% RSLogix 500 project project4.RSS, saved by version 8.30.00.16 %
PROJECT "UNTITLED"    % processor: Bul.1763 MicroLogix 1100 Series B %

PROGRAM FILES
  LAD 2 "MAIN"  4 rungs
  LAD 3 "DIGITAL IO"  7 rungs
  LAD 4 "CONTROLS"  13 rungs
  LAD 5 "MODES"  8 rungs

DATA FILES
  O0 OUTPUT  5 elements
  I1 INPUT  7 elements
  S2 STATUS  66 elements
  B3 BINARY  2 elements
  T4 TIMER  3 elements
  C5 COUNTER  1 elements
  R6 CONTROL  1 elements
  N7 INTEGER  2 elements
  F8 FLOAT  1 elements

LADDER 2 "MAIN"
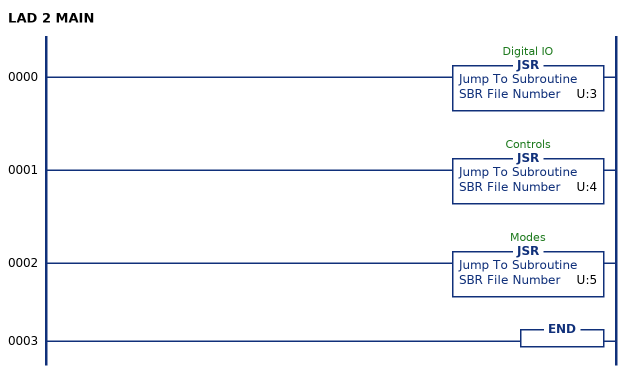
% Rung: 0 %
SOR JSR U:3 EOR
%   U:3  "Digital IO" %
% Rung: 1 %
SOR JSR U:4 EOR
%   U:4  "Controls" %
% Rung: 2 %
SOR JSR U:5 EOR
%   U:5  "Modes" %
% Rung: 3 %
SOR END EOR

LADDER 3 "DIGITAL IO"
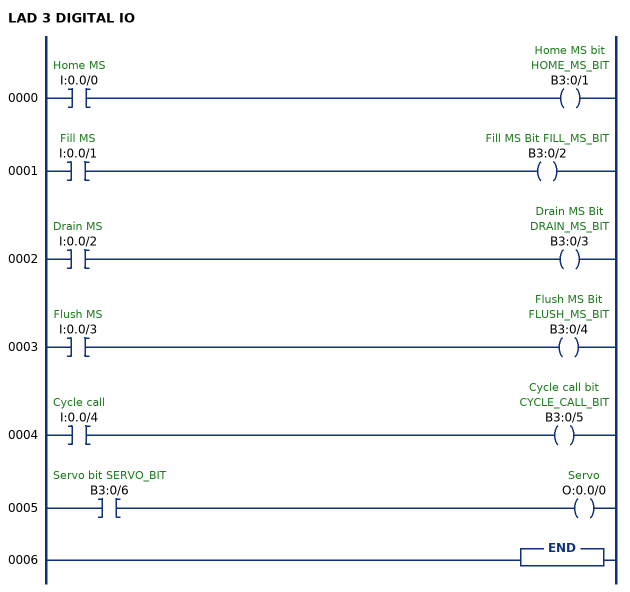
% Rung: 0 %
SOR XIC I:0.0/0 OTE B3:0/1 EOR
%   I:0.0/0  "Home MS" %
%   B3:0/1  HOME_MS_BIT  "Home MS bit" %
% Rung: 1 %
SOR XIC I:0.0/1 OTE B3:0/2 EOR
%   I:0.0/1  "Fill MS" %
%   B3:0/2  FILL_MS_BIT  "Fill MS Bit" %
% Rung: 2 %
SOR XIC I:0.0/2 OTE B3:0/3 EOR
%   I:0.0/2  "Drain MS" %
%   B3:0/3  DRAIN_MS_BIT  "Drain MS Bit" %
% Rung: 3 %
SOR XIC I:0.0/3 OTE B3:0/4 EOR
%   I:0.0/3  "Flush MS" %
%   B3:0/4  FLUSH_MS_BIT  "Flush MS Bit" %
% Rung: 4 %
SOR XIC I:0.0/4 OTE B3:0/5 EOR
%   I:0.0/4  "Cycle call" %
%   B3:0/5  CYCLE_CALL_BIT  "Cycle call bit" %
% Rung: 5 %
SOR XIC B3:0/6 OTE O:0.0/0 EOR
%   B3:0/6  SERVO_BIT  "Servo bit" %
%   O:0.0/0  "Servo" %
% Rung: 6 %
SOR END EOR

LADDER 4 "CONTROLS"
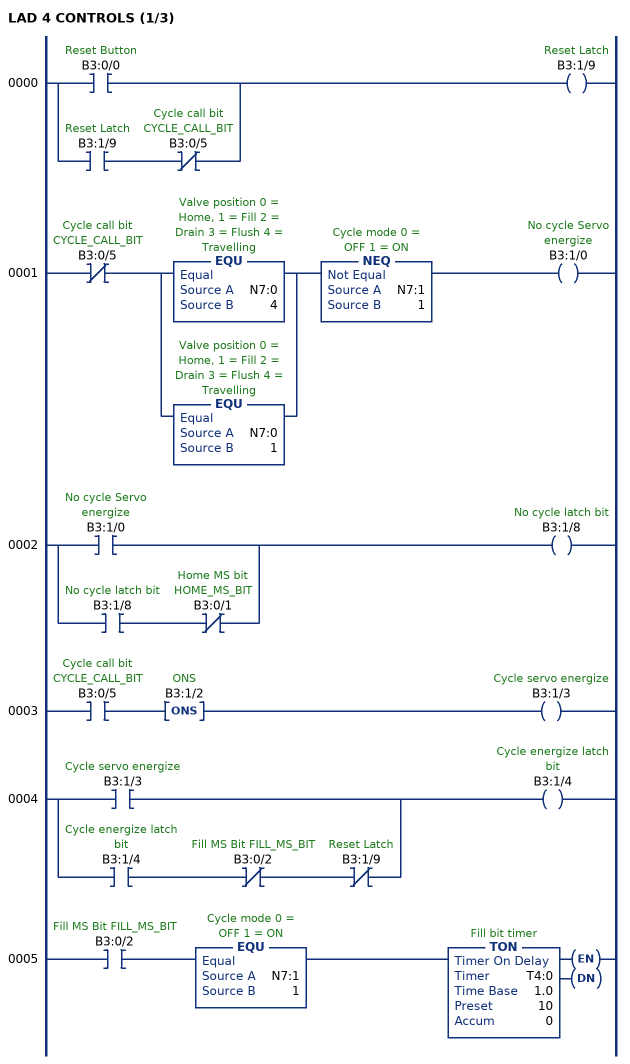
% Rung: 0 %
SOR BST XIC B3:0/0 NXB XIC B3:1/9 XIO B3:0/5 BND OTE B3:1/9 EOR
%   B3:0/0  "Reset Button" %
%   B3:1/9  "Reset Latch" %
%   B3:0/5  CYCLE_CALL_BIT  "Cycle call bit" %
% Rung: 1 %
SOR XIO B3:0/5 BST EQU N7:0 4 NXB EQU N7:0 1 BND NEQ N7:1 1 OTE B3:1/0 EOR
%   B3:0/5  CYCLE_CALL_BIT  "Cycle call bit" %
%   N7:0  "Valve position 0 = Home, 1 = Fill 2 = Drain 3 = Flush 4 = Travelling" %
%   N7:1  "Cycle mode 0 = OFF 1 = ON" %
%   B3:1/0  "No cycle Servo energize" %
% Rung: 2 %
SOR BST XIC B3:1/0 NXB XIC B3:1/8 XIO B3:0/1 BND OTE B3:1/8 EOR
%   B3:1/0  "No cycle Servo energize" %
%   B3:1/8  "No cycle latch bit" %
%   B3:0/1  HOME_MS_BIT  "Home MS bit" %
% Rung: 3 %
SOR XIC B3:0/5 ONS B3:1/2 OTE B3:1/3 EOR
%   B3:0/5  CYCLE_CALL_BIT  "Cycle call bit" %
%   B3:1/2  "ONS" %
%   B3:1/3  "Cycle servo energize" %
% Rung: 4 %
SOR BST XIC B3:1/3 NXB XIC B3:1/4 XIO B3:0/2 XIO B3:1/9 BND OTE B3:1/4 EOR
%   B3:1/3  "Cycle servo energize" %
%   B3:1/4  "Cycle energize latch bit" %
%   B3:0/2  FILL_MS_BIT  "Fill MS Bit" %
%   B3:1/9  "Reset Latch" %
% Rung: 5 %
SOR XIC B3:0/2 EQU N7:1 1 TON T4:0 1.0 10 0 EOR
%   B3:0/2  FILL_MS_BIT  "Fill MS Bit" %
%   N7:1  "Cycle mode 0 = OFF 1 = ON" %
%   T4:0  "Fill bit timer" %

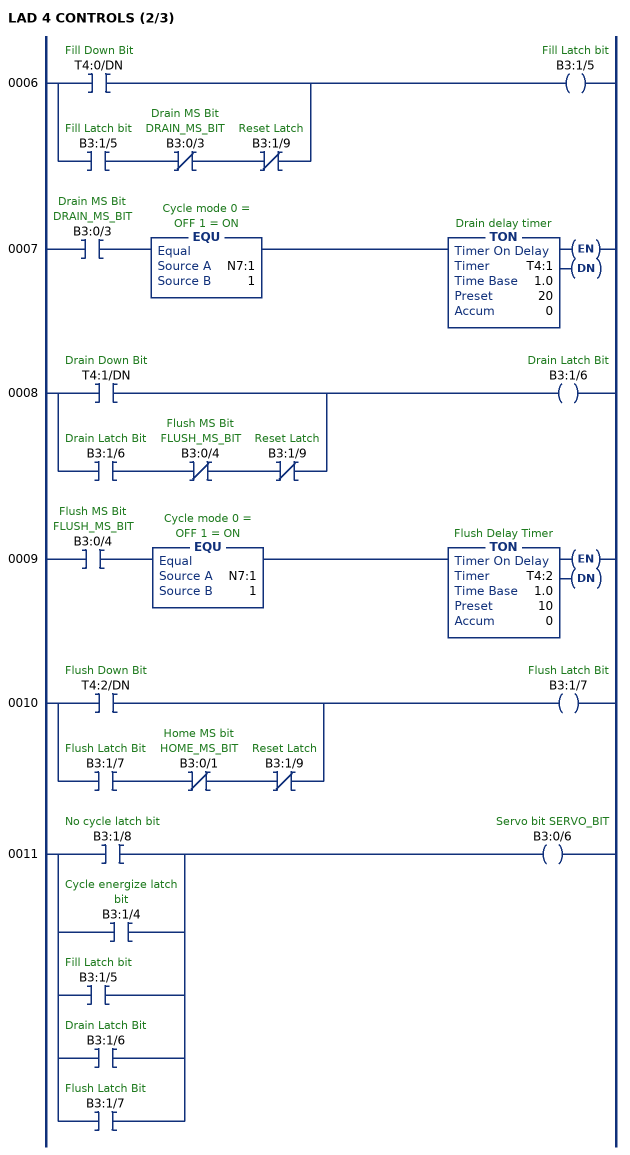
% Rung: 6 %
SOR BST XIC T4:0/DN NXB XIC B3:1/5 XIO B3:0/3 XIO B3:1/9 BND OTE B3:1/5 EOR
%   T4:0/DN  "Fill Down Bit" %
%   B3:1/5  "Fill Latch bit" %
%   B3:0/3  DRAIN_MS_BIT  "Drain MS Bit" %
%   B3:1/9  "Reset Latch" %
% Rung: 7 %
SOR XIC B3:0/3 EQU N7:1 1 TON T4:1 1.0 20 0 EOR
%   B3:0/3  DRAIN_MS_BIT  "Drain MS Bit" %
%   N7:1  "Cycle mode 0 = OFF 1 = ON" %
%   T4:1  "Drain delay timer" %
% Rung: 8 %
SOR BST XIC T4:1/DN NXB XIC B3:1/6 XIO B3:0/4 XIO B3:1/9 BND OTE B3:1/6 EOR
%   T4:1/DN  "Drain Down Bit" %
%   B3:1/6  "Drain Latch Bit" %
%   B3:0/4  FLUSH_MS_BIT  "Flush MS Bit" %
%   B3:1/9  "Reset Latch" %
% Rung: 9 %
SOR XIC B3:0/4 EQU N7:1 1 TON T4:2 1.0 10 0 EOR
%   B3:0/4  FLUSH_MS_BIT  "Flush MS Bit" %
%   N7:1  "Cycle mode 0 = OFF 1 = ON" %
%   T4:2  "Flush Delay Timer" %
% Rung: 10 %
SOR BST XIC T4:2/DN NXB XIC B3:1/7 XIO B3:0/1 XIO B3:1/9 BND OTE B3:1/7 EOR
%   T4:2/DN  "Flush Down Bit" %
%   B3:1/7  "Flush Latch Bit" %
%   B3:0/1  HOME_MS_BIT  "Home MS bit" %
%   B3:1/9  "Reset Latch" %
% Rung: 11 %
SOR BST XIC B3:1/8 NXB XIC B3:1/4 NXB XIC B3:1/5 NXB XIC B3:1/6 NXB XIC B3:1/7 BND OTE B3:0/6 EOR
%   B3:1/8  "No cycle latch bit" %
%   B3:1/4  "Cycle energize latch bit" %
%   B3:1/5  "Fill Latch bit" %
%   B3:1/6  "Drain Latch Bit" %
%   B3:1/7  "Flush Latch Bit" %
%   B3:0/6  SERVO_BIT  "Servo bit" %

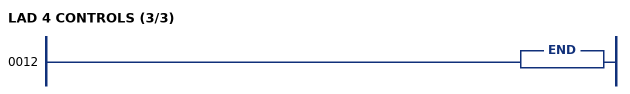
% Rung: 12 %
SOR END EOR

LADDER 5 "MODES"
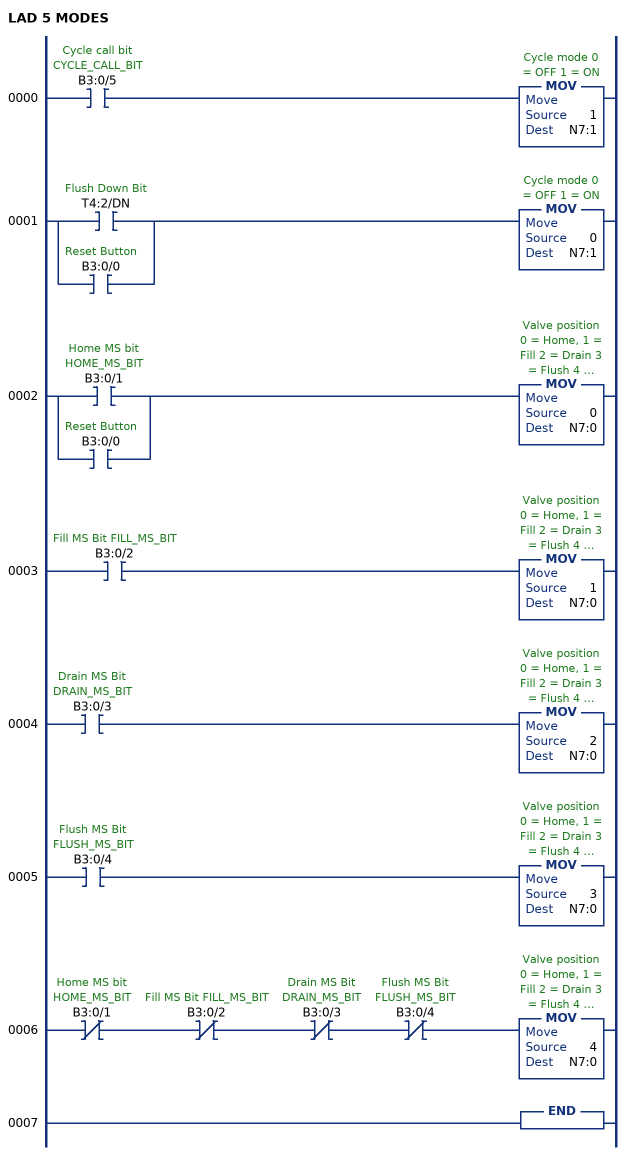
% Rung: 0 %
SOR XIC B3:0/5 MOV 1 N7:1 EOR
%   B3:0/5  CYCLE_CALL_BIT  "Cycle call bit" %
%   N7:1  "Cycle mode 0 = OFF 1 = ON" %
% Rung: 1 %
SOR BST XIC T4:2/DN NXB XIC B3:0/0 BND MOV 0 N7:1 EOR
%   T4:2/DN  "Flush Down Bit" %
%   B3:0/0  "Reset Button" %
%   N7:1  "Cycle mode 0 = OFF 1 = ON" %
% Rung: 2 %
SOR BST XIC B3:0/1 NXB XIC B3:0/0 BND MOV 0 N7:0 EOR
%   B3:0/1  HOME_MS_BIT  "Home MS bit" %
%   B3:0/0  "Reset Button" %
%   N7:0  "Valve position 0 = Home, 1 = Fill 2 = Drain 3 = Flush 4 = Travelling" %
% Rung: 3 %
SOR XIC B3:0/2 MOV 1 N7:0 EOR
%   B3:0/2  FILL_MS_BIT  "Fill MS Bit" %
%   N7:0  "Valve position 0 = Home, 1 = Fill 2 = Drain 3 = Flush 4 = Travelling" %
% Rung: 4 %
SOR XIC B3:0/3 MOV 2 N7:0 EOR
%   B3:0/3  DRAIN_MS_BIT  "Drain MS Bit" %
%   N7:0  "Valve position 0 = Home, 1 = Fill 2 = Drain 3 = Flush 4 = Travelling" %
% Rung: 5 %
SOR XIC B3:0/4 MOV 3 N7:0 EOR
%   B3:0/4  FLUSH_MS_BIT  "Flush MS Bit" %
%   N7:0  "Valve position 0 = Home, 1 = Fill 2 = Drain 3 = Flush 4 = Travelling" %
% Rung: 6 %
SOR XIO B3:0/1 XIO B3:0/2 XIO B3:0/3 XIO B3:0/4 MOV 4 N7:0 EOR
%   B3:0/1  HOME_MS_BIT  "Home MS bit" %
%   B3:0/2  FILL_MS_BIT  "Fill MS Bit" %
%   B3:0/3  DRAIN_MS_BIT  "Drain MS Bit" %
%   B3:0/4  FLUSH_MS_BIT  "Flush MS Bit" %
%   N7:0  "Valve position 0 = Home, 1 = Fill 2 = Drain 3 = Flush 4 = Travelling" %
% Rung: 7 %
SOR END EOR

OTHER DOCUMENTED ADDRESSES
  B3:1/1  "ONS"

DATA TABLE (non-zero values as saved)
DATA T4
% .PRE .ACC %
% T4:0 % 10 0
% T4:1 % 20 0
% T4:2 % 10 0
